FUNCTION_BLOCK EL4024
VAR
	_io : EL4xx4_Data;
	{attribute addProperty Name "WcState"}
	_wcState : WcStateBase;
	{attribute addProperty Name "Info data"}
	_infoData : InfoDataAds;
END_VAR

PROPERTY IO : REFERENCE TO EL4xx4_Data
GET
IO REF= _io;
END_GET
END_PROPERTY

PROPERTY WcState : REFERENCE TO WcStateBase
GET
WcState REF= _wcState;
END_GET
END_PROPERTY

END_FUNCTION_BLOCK

(* stored: Version 1.1.0.1, ProductVersion 3.1.4024.9
   POU EL4024: Id {3a58983b-98e3-07f0-04c6-0bf057321dd3}, SpecialFunc None
   Property IO: Id {a7b781ae-fa84-04d4-16a2-5931db11e3b3}
   Get Get: Id {15c70dcd-1dcf-064a-13eb-8e587511449b}
   Property WcState: Id {c5d48162-b511-0b4f-0d3e-be8fd40e5fb9}
   Get Get: Id {1eca8211-eedb-0415-2cc9-2f4790e70c1d} *)
